// TIA Portal V20 export
TYPE "TypeLinmotSd"
   STRUCT
      Ctrl : Struct   // control word
         SwitchOn : Bool;   // 0 = A-Stop, -> Current = 0, power switches disabled
         VoltageEnable : Bool;   // 0 = Power switches disabled without microcontroller action
         QuickStop : Bool;   // 0 = Quick Stop -> Current = 0 -> H-Bridges disabled
         EnableOperation : Bool;   // Position controller active Motion Commands enabled
         Abort : Bool;   // 0 = Quick Stop position control rests active, motion
         Freeze : Bool;   // 0 = Quick Stop position control rests active, Target position
         GoToPosition : Bool;   // 1 = Go to fixed parameterized Position. Wait for release of signal
         ErrorAcknoledge : Bool;   // 1 = Rising edge of signal acknowledges error
         JogMovePlus : Bool;   // 1 = Jog Move +
         JogMoveMinus : Bool;   // 1 = Jog Move -
         SpecialMove : Bool;   // 1 = Special Mode
         Home : Bool;   // 1 = At startup bit 11 Status word is cleared, until procedure
         ClearanceCheck : Bool;   // 1 = Enable Clearance Check Movement
         GoToInitialPosition : Bool;   // 1 = Rising edge will start go to initial position
         Linearizing : Bool;   // Reserved
         PhaseSearch : Bool;   // 1 = Enable Phase Search Movements
      END_STRUCT;
      McHd : Struct   // motion command header
         CC0 : Bool;   // Command Count bit 0
         CC1 : Bool;   // Command Count bit 1
         CC2 : Bool;   // Command Count bit 2
         CC3 : Bool;   // Command Count bit 3
         SubID0 : Bool;   // Sub ID bit 0
         SubID1 : Bool;   // Sub ID bit 1
         SubID2 : Bool;   // Sub ID bit 2
         SubID3 : Bool;   // Sub ID bit 3
         MasterID : Byte;   // Master ID
      END_STRUCT;
      McPar1 : DInt;   // motion command parameter 1
      McPar2 : DInt;   // motion command parameter 2
      McPar3 : DInt;   // motion command parameter 3
      McPar4 : DInt;   // motion command parameter 4
      McPar5 : DInt;   // motion command parameter 5
      CgfHd : Int;   // Config Header
      CfgId : Int;   // Config Index
      CfgVal : DInt;   // Config Value
   END_STRUCT;
END_TYPE
